// TIA Portal V17 export
// export: Created 2025-06-26T06:49:13.096488Z, ExportSetting WithDefaults, DisplayName Totally Integrated Automation Portal, DisplayVersion V17 Update 8, DisplayName TIA Portal Openness, DisplayVersion V17 Update 8, DisplayName TIA Portal Version Control Interface, DisplayVersion V17, DisplayName STEP 7 Professional, DisplayVersion V17 Update 8, DisplayName STEP 7 Safety, DisplayVersion V17 Update 6, DisplayName WinCC Advanced, DisplayVersion V17 Update 8
FUNCTION_BLOCK "ValveControl"   // FB27, FBD
TITLE = Setpoint selection & drivers
{ S7_Optimized_Access := 'TRUE' }
VERSION : 0.1
// stored: AutoNumber true, IsIECCheckEnabled false, IsRetainMemResEnabled false, MemoryReserve 100, SetENOAutomatically false, UDAEnableTagReadback false
   VAR_INPUT
      ValveSetpoint { ExternalAccessible := 'False'; ExternalVisible := 'False'; ExternalWritable := 'False'} : Real;   // [%] Valve position from regulator
   END_VAR
   VAR
      Setpoint { ExternalAccessible := 'False'; ExternalVisible := 'False'; ExternalWritable := 'False'} : Real;   // [%] Selected valve position
   END_VAR
   VAR_TEMP   // added for the SCL form of the ladder/FBD networks
      _w1 : Bool;
      _w2 : Bool;
   END_VAR
BEGIN

REGION Network 1 (SCL): Comment & history
   // Run valve drivers and do any switching of setpoints in case a valve is part of more than one control axis
END_REGION

REGION Network 2: Expansion valves
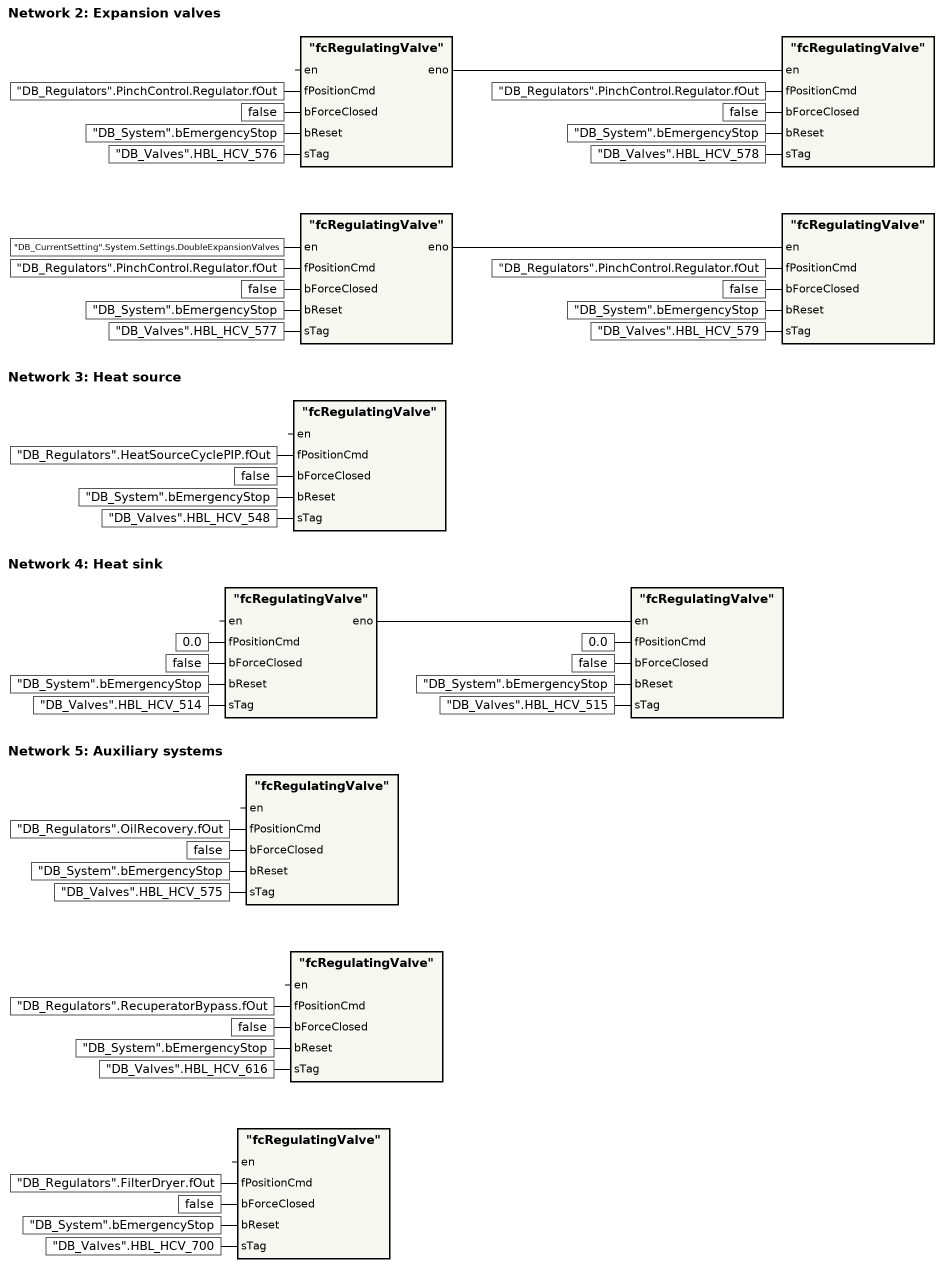
   "fcRegulatingValve"(fPositionCmd := "DB_Regulators".PinchControl.Regulator.fOut,
                       bForceClosed := false,
                       bReset := "DB_System".bEmergencyStop,
                       sTag := "DB_Valves".HBL_HCV_576,
                       ENO => #_w1);
   IF #_w1 THEN
       "fcRegulatingValve"(fPositionCmd := "DB_Regulators".PinchControl.Regulator.fOut,
                           bForceClosed := false,
                           bReset := "DB_System".bEmergencyStop,
                           sTag := "DB_Valves".HBL_HCV_578);
   END_IF;
   "fcRegulatingValve"(EN := "DB_CurrentSetting".System.Settings.DoubleExpansionValves,
                       fPositionCmd := "DB_Regulators".PinchControl.Regulator.fOut,
                       bForceClosed := false,
                       bReset := "DB_System".bEmergencyStop,
                       sTag := "DB_Valves".HBL_HCV_577,
                       ENO => #_w2);
   IF #_w2 THEN
       "fcRegulatingValve"(fPositionCmd := "DB_Regulators".PinchControl.Regulator.fOut,
                           bForceClosed := false,
                           bReset := "DB_System".bEmergencyStop,
                           sTag := "DB_Valves".HBL_HCV_579);
   END_IF;
END_REGION

REGION Network 3: Heat source
   "fcRegulatingValve"(fPositionCmd := "DB_Regulators".HeatSourceCyclePIP.fOut,
                       bForceClosed := false,
                       bReset := "DB_System".bEmergencyStop,
                       sTag := "DB_Valves".HBL_HCV_548);
END_REGION

REGION Network 4: Heat sink
   "fcRegulatingValve"(fPositionCmd := 0.0,
                       bForceClosed := false,
                       bReset := "DB_System".bEmergencyStop,
                       sTag := "DB_Valves".HBL_HCV_514,
                       ENO => #_w1);
   IF #_w1 THEN
       "fcRegulatingValve"(fPositionCmd := 0.0,
                           bForceClosed := false,
                           bReset := "DB_System".bEmergencyStop,
                           sTag := "DB_Valves".HBL_HCV_515);
   END_IF;
END_REGION

REGION Network 5: Auxiliary systems
   "fcRegulatingValve"(fPositionCmd := "DB_Regulators".OilRecovery.fOut,
                       bForceClosed := false,
                       bReset := "DB_System".bEmergencyStop,
                       sTag := "DB_Valves".HBL_HCV_575);
   "fcRegulatingValve"(fPositionCmd := "DB_Regulators".RecuperatorBypass.fOut,
                       bForceClosed := false,
                       bReset := "DB_System".bEmergencyStop,
                       sTag := "DB_Valves".HBL_HCV_616);
   "fcRegulatingValve"(fPositionCmd := "DB_Regulators".FilterDryer.fOut,
                       bForceClosed := false,
                       bReset := "DB_System".bEmergencyStop,
                       sTag := "DB_Valves".HBL_HCV_700);
END_REGION
END_FUNCTION_BLOCK
